{attribute 'reflection'}
FUNCTION_BLOCK ABSTRACT FB_Object IMPLEMENTS I_Object
VAR
    _nIdentity:         ULINT;
    _ipParent:          I_Object;

    {attribute 'instance-path'}
    {attribute 'noinit'}
    _sPath:             STRING(MAX_STRING_LENGTH);
END_VAR

PROPERTY bOrphan : BOOL
GET
bOrphan := THIS^._ipParent = 0;
END_GET
END_PROPERTY

METHOD EqualsTo : BOOL
VAR_INPUT
    ipComparedObject:           I_Object;
END_VAR
IF ipComparedObject.nIdentity <> 0 THEN
    EqualsTo := ipComparedObject.nIdentity = THIS^._nIdentity;
END_IF
END_METHOD

METHOD FB_init : BOOL
VAR_INPUT
    bInitRetains:           BOOL; // if TRUE, the retain variables are initialized (warm start / cold start)
    bInCopyCode:            BOOL;  // if TRUE, the instance afterwards gets moved into the copy code (online change)
    ipParentObject:         I_Object;
END_VAR
_nIdentity := ADR(THIS^);
_ipParent := ipParentObject;
END_METHOD

PROPERTY ipContext : I_Context
GET
IF NOT THIS^.bOrphan THEN
    ipContext := THIS^.ipParent.ipContext;
END_IF
END_GET
END_PROPERTY

PROPERTY ipParent : I_Object
GET
IF _ipParent <> 0 THEN
    ipParent := THIS^._ipParent;
    RETURN;
END_IF
END_GET
END_PROPERTY

PROPERTY nIdentity : ULINT
GET
THIS^._nIdentity := ADR(THIS^);
nIdentity := THIS^._nIdentity;
END_GET
END_PROPERTY

PROPERTY sPath : STRING(MAX_STRING_LENGTH)
GET
sPath := THIS^._sPath;
END_GET
END_PROPERTY

END_FUNCTION_BLOCK

(* stored: Version 1.1.0.1, ProductVersion 3.1.4024.12
   POU FB_Object: Id {87ccbc5a-8a98-4cc4-aa55-78ff92f7c37f}, SpecialFunc None
   Property bOrphan: Id {b322e367-c154-402e-88b0-f0f448e22ea7}
   Get Get: Id {37a6e89f-2a4c-4eec-9652-407a301a9ce5}
   Method EqualsTo: Id {e0d9c976-b19a-4134-8e2d-cb5c401117cc}
   Method FB_init: Id {058b6abe-0386-4ead-9210-33fdf22e4732}
   Property ipContext: Id {af011723-3225-42bc-a3cf-ab5677defbfe}
   Get Get: Id {40949f99-26a3-42b6-8031-091b2b3252b0}
   Property ipParent: Id {476836f0-75a2-440a-a857-bf17b0a7f0dc}
   Get Get: Id {07e655a1-6465-4a2f-826a-bf0c292f7655}
   Property nIdentity: Id {f3f9b85a-2c87-4f9c-bb99-0511480c45ad}
   Get Get: Id {a92d2096-f26b-4a48-9f10-1d6a8572e4ae}
   Property sPath: Id {57079563-ab74-4c88-ae4d-a3108deae837}
   Get Get: Id {29f1b486-0a4c-4485-afe9-f9913d8160f7} *)
